Staubli VAL3: computeFrame.pgx

public program computeFrame(num x_nNewFrame)
  local num i
begin
    // recompute all the point into the new frame
  for i=0 to size(pEditPoint.tData)-1
    pEditPoint.tData[i].pPoint.trsf=position(pEditPoint.tData[i].pPoint,saveData:fFrameItem[x_nNewFrame].fFrame)
  endFor
end
